FUNCTION_BLOCK FB_MaintainLaserOperation EXTENDS FB_Operation
VAR_INPUT
END_VAR
VAR_OUTPUT
	q_bShutdownLaser : BOOL;
END_VAR
VAR
END_VAR

// Let FB_Operation do its thing 
SUPER^(iq_sMessageBuffer := iq_sMessageBuffer);

METHOD PROTECTED M_AllTransportTubeValvesClosed : BOOL
VAR_INPUT
END_VAR
VAR
	nIter : UINT;
	eTT : T_TransportTube;
	fbTT : REFERENCE TO FB_TransportTube;
END_VAR
M_AllTransportTubeValvesClosed := TRUE;

FOR nIter := 1 TO GVL_TransportTubes.NUM_TRANSPORT_TUBES DO
	eTT := GVL_TransportTubes.aTubes[nIter];
	fbTT REF= F_GetTransportTube(eTT);

	IF NOT fbTT.q_stConfig.stDevices.refGateValve.M_IsClosed() THEN
		M_AllTransportTubeValvesClosed := FALSE;
		RETURN;
	END_IF
END_FOR
END_METHOD

METHOD PROTECTED M_CloseAllTransportTubeValves
VAR_INPUT
END_VAR
VAR
	nIter : UINT;
	eTT : T_TransportTube;
	fbTT : REFERENCE TO FB_TransportTube;
END_VAR
FOR nIter := 1 TO GVL_TransportTubes.NUM_TRANSPORT_TUBES DO
	eTT := GVL_TransportTubes.aTubes[nIter];
	fbTT REF= F_GetTransportTube(eTT);

	fbTT.q_stConfig.stDevices.refGateValve.M_Set_OPN_SW(FALSE);
END_FOR
END_METHOD

METHOD PROTECTED M_FatalError
VAR_INPUT
	i_ErrorMessage : STRING;
END_VAR
SUPER^.M_FatalError(i_ErrorMessage);
M_ShutdownLaser();
END_METHOD

METHOD PUBLIC M_ResetError
VAR_INPUT
END_VAR
SUPER^.M_ResetError();
q_bShutdownLaser := FALSE;
END_METHOD

METHOD PROTECTED M_ShutdownLaser
VAR_INPUT
END_VAR
q_bShutdownLaser := TRUE;
END_METHOD

END_FUNCTION_BLOCK

(* stored: Version 1.1.0.1, ProductVersion 3.1.4022.17
   POU FB_MaintainLaserOperation: Id {01f4e0f9-508d-4564-920a-841ec286a4bd}, SpecialFunc None
   Method M_AllTransportTubeValvesClosed: Id {ccc571c6-4175-48f1-8d3e-bdd491494d87}
   Method M_CloseAllTransportTubeValves: Id {f0574d64-0945-4a16-96d0-702f95d9f806}
   Method M_FatalError: Id {3e3c79d9-a8f3-419e-a59c-ac88697e8597}
   Method M_ResetError: Id {c086e734-a4ca-4ff5-a730-57ac81287e91}
   Method M_ShutdownLaser: Id {665d0026-87e9-4768-8d69-0114183a526c} *)
